FUNCTION_BLOCK CountOfElements (* Returns the lower bound of the dimension of the given array *)
  (* Function: inspired by Siemens: CountOfElements; Description: Copyright (c) 2026 Demmler Andreas Fahrzeugbau This program and the accompanying materials are made available under the terms of the Eclipse Public License 2.0 which is available at https://www.eclipse.org/legal/epl-2.0/ SPDX-License-Identifier: EPL-2.0 *)
  (* Version 1.0, 2026-01-23, Franz Höpfninger, Demmler Andreas Fahrzeugbau, Initial Implementation *)
  PACKAGE eclipse4diac::convert;
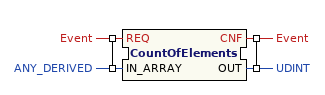
  EVENT_INPUT
    REQ WITH IN_ARRAY; (* Service Request *)
  END_EVENT
  EVENT_OUTPUT
    CNF WITH OUT; (* Confirmation of Requested Service *)
  END_EVENT
  VAR_INPUT
    IN_ARRAY : ANY_DERIVED; (* input array *)
  END_VAR
  VAR_OUTPUT
    OUT : UDINT; (* Number of Elements in the Array *)
  END_VAR
END_FUNCTION_BLOCK
